TYPE TYP_VALVE_POS_HW :
STRUCT
	ReachedHP AT %I* : BOOL;
	ReachedWP AT %I* : BOOL;
END_STRUCT
END_TYPE

(* stored: Version 1.1.0.1, ProductVersion 3.1.4024.12
   DUT TYP_VALVE_POS_HW: Id {9fab6ea9-0be1-411c-b205-ca1b03436ffa} *)
